{attribute 'OPC.UA.DA.StructuredType' := '1'}
TYPE stOB :
STRUCT
	sName		: STRING[10];
	uliOrder	: ULINT;
	xFull		: BOOL;
	xEmpty		: BOOL;
	xAvailable	: BOOL;
	xEnable		: BOOL;
END_STRUCT
END_TYPE

(* stored: Version 1.1.0.1, ProductVersion 3.1.4024.11
   DUT stOB: Id {1ba2abcf-9b3b-4d89-91eb-f58482078643} *)
